KUKA KRL program: Bolge_3_Palet_Ort.src, Bolge_3_Palet_Ort.dat

--- Bolge_3_Palet_Ort.src ---
&ACCESS RVP1
&REL 44
&PARAM DISKPATH = KRC:\R1\Program\Sub_Rutinler
DEF  Bolge_3_Palet_Ort ( )
;FOLD INI;%{PE}
  ;FOLD BASISTECH INI
    GLOBAL INTERRUPT DECL 3 WHEN $STOPMESS==TRUE DO IR_STOPM ( )
    INTERRUPT ON 3
    BAS (#INITMOV,0 )
  ;ENDFOLD (BASISTECH INI)
  ;FOLD USER INI
    ;Make your modifications here

  ;ENDFOLD (USER INI)
;ENDFOLD (INI)



;;FOLD PTP B3_MASTER CONT Vel=100 % PDAT1 Tool[1]:Gripper Base[0] ;%{PE}
;;FOLD Parameters ;%{h}
;;Params IlfProvider=kukaroboter.basistech.inlineforms.movement.old; Kuka.IsGlobalPoint=False; Kuka.PointName=B3_MASTER; Kuka.BlendingEnabled=True; Kuka.MoveDataPtpName=PDAT1; Kuka.VelocityPtp=100; Kuka.CurrentCDSetIndex=0; Kuka.MovementParameterFieldEnabled=True; IlfCommand=PTP
;;ENDFOLD
;$BWDSTART = FALSE
;PDAT_ACT = PPDAT1
;FDAT_ACT = FB3_MASTER
;BAS(#PTP_PARAMS, 100.0)
;SET_CD_PARAMS (0)
;PTP XB3_MASTER C_Dis
;;ENDFOLD


PaletMasterX=1840
PaletMasterY=1240


Base_Data[3]=Frame_Donustur(XB3_MASTER)
BASE_DATA[3].x=BASE_DATA[3].x-(PaletMasterX/2)
BASE_DATA[3].Y=BASE_DATA[3].Y+(PaletMasterY/2)

      IF (ParcaUzunluk<=1500)THEN

         BASE_DATA[3].x=BASE_DATA[3].x+(PaletUzunluk/2)
         BASE_DATA[3].Y=BASE_DATA[3].Y-(PaletGenislik/2)

      ENDIF

      IF (ParcaUzunluk>=1600) AND (ParcaUzunluk<=3000) THEN

         BASE_DATA[3].x=BASE_DATA[3].x+(PaletUzunluk/2)

         BASE_DATA[3].Y=BASE_DATA[3].Y-(PaletGenislik/2)

      ENDIF

END
DEFFCT FRAME Frame_Donustur(e6GeciciPos:IN)
   ;FOLD  Tanimlamalar
      DECL E6POS e6GeciciPos
      DECL FRAME ReturnFrame
   ;ENDFOLD
   ReturnFrame=$Nullframe
   ReturnFrame.X=e6GeciciPos.X
   ReturnFrame.Y=e6GeciciPos.Y
   ReturnFrame.Z=e6GeciciPos.Z
   ReturnFrame.A=e6GeciciPos.A
   ReturnFrame.B=e6GeciciPos.B
   ReturnFrame.C=e6GeciciPos.C
   RETURN ReturnFrame
ENDFCT

--- Bolge_3_Palet_Ort.dat ---
&ACCESS  RVP
&PARAM DISKPATH = KRC:\R1\Program\Sub_Rutinler
&REL 42
DEFDAT  BOLGE_3_PALET_ORT
;FOLD EXTERNAL DECLARATIONS;%{PE}%MKUKATPBASIS,%CEXT,%VCOMMON,%P
;FOLD BASISTECH EXT;%{PE}%MKUKATPBASIS,%CEXT,%VEXT,%P
EXT  BAS (BAS_COMMAND  :IN,REAL  :IN )
DECL INT SUCCESS
;ENDFOLD (BASISTECH EXT)
;FOLD USER EXT;%{E}%MKUKATPUSER,%CEXT,%VEXT,%P
;Make your modifications here

;ENDFOLD (USER EXT)
;ENDFOLD (EXTERNAL DECLARATIONS)
DECL E6POS XB3_MASTER={X 1194.49854,Y -2009.09937,Z -1230.98389,A -0.338213325,B -9.00781846E-15,C -3.05002443E-12,S 2,T 2,E1 0.0,E2 0.0,E3 0.0,E4 0.0,E5 0.0,E6 0.0}
DECL FDAT FB3_MASTER={TOOL_NO 1,BASE_NO 0,IPO_FRAME #BASE,POINT2[] " "}
DECL PDAT PPDAT1={VEL 100.000,ACC 100.000,APO_DIST 500.000,APO_MODE #CDIS,GEAR_JERK 100.000,EXAX_IGN 0}
DECL MODULEPARAM_T LAST_TP_PARAMS={PARAMS[] "Kuka.VelocityFieldEnabled=True; Kuka.ColDetectFieldEnabled=True; Kuka.MovementParameterFieldEnabled=True; Kuka.IsAngleEnabled=False; Kuka.PointName=B3_MASTER; Kuka.FrameData.base_no=0; Kuka.FrameData.tool_no=1; Kuka.FrameData.ipo_frame=#BASE; Kuka.FrameData.point2=; Kuka.isglobalpoint=False; Kuka.MoveDataPtpName=PDAT1; Kuka.MovementDataPdat.apo_mode=#CDIS; Kuka.MovementDataPdat.apo_dist=500; Kuka.MovementData.vel=100; Kuka.MovementData.acc=100; Kuka.MovementData.exax_ign=0; Kuka.VelocityPtp=100; Kuka.BlendingEnabled=True; Kuka.APXEnabled=False; Kuka.CurrentCDSetIndex=0   "}
ENDDAT
